Staubli VAL3: resetSignal.pgx

program resetSignal(bool x_bCondition (dimensions=1), dio x_doSignal (dimensions=1))
begin
  if x_bCondition
    if x_doSignal==true
      x_doSignal=false
    endIf
  endIf
end
